// Mitsubishi GX Works2 project: BookEX6_14 Bistable   PLC: Q13UDV

// global labels: Global
VAR_GLOBAL
  bVar0 AT M5000 : BOOL;
  abArray0 AT M5010 : ARRAY [0..49] OF BOOL;
  sStr0 AT D5000 : STRING[199];
  sStr1 AT D5100 : STRING[199];
  sStr2 AT D5200 : STRING[199];
  sStr3 AT D5300 : STRING[199];
  sStr4 AT D5400 : STRING[199];
  sStr5 AT D5500 : STRING[199];
  sStr6 AT D5600 : STRING[199];
  sStr7 AT D5700 : STRING[199];
  sStr8 AT D5800 : STRING[199];
  sStr9 AT D5900 : STRING[199];
  iVar0 AT D4500 : INT;
  iVar1 AT D4501 : INT;
  iVar2 AT D4502 : INT;
  iVar3 AT D4503 : INT;
  iVar4 AT D4504 : INT;
  iVar5 AT D4505 : INT;
  iVar6 AT D4506 : INT;
  iVar7 AT D4507 : INT;
  iVar8 AT D4508 : INT;
  iVar9 AT D4509 : INT;
  dVar0 AT D4510 : DINT;
  dVar1 AT D4512 : DINT;
  dVar2 AT D4514 : DINT;
  dVar3 AT D4516 : DINT;
  dVar4 AT D4518 : DINT;
  dVar5 AT D4520 : DINT;
  dVar6 AT D4522 : DINT;
  dVar7 AT D4524 : DINT;
  dVar8 AT D4526 : DINT;
  dVar9 AT D4528 : DINT;
  wVar0 AT D4530 : WORD;
  wVar1 AT D4531 : WORD;
  wVar2 AT D4532 : WORD;
  wVar3 AT D4533 : WORD;
  wVar4 AT D4534 : WORD;
  wVar5 AT D4535 : WORD;
  wVar6 AT D4536 : WORD;
  wVar7 AT D4537 : WORD;
  wVar8 AT D4538 : WORD;
  wVar9 AT D4539 : WORD;
  dwVar0 AT D4540 : DWORD;
  dwVar1 AT D4542 : DWORD;
  dwVar2 AT D4544 : DWORD;
  dwVar3 AT D4546 : DWORD;
  dwVar4 AT D4548 : DWORD;
  dwVar5 AT D4550 : DWORD;
  dwVar6 AT D4552 : DWORD;
  dwVar7 AT D4554 : DWORD;
  dwVar8 AT D4556 : DWORD;
  dwVar9 AT D4558 : DWORD;
  fsVar0 AT D4560 : REAL;
  fsVar1 AT D4562 : REAL;
  fsVar2 AT D4564 : REAL;
  fsVar3 AT D4566 : REAL;
  fsVar4 AT D4568 : REAL;
  fsVar5 AT D4570 : REAL;
  fsVar6 AT D4572 : REAL;
  fsVar7 AT D4574 : REAL;
  fsVar8 AT D4576 : REAL;
  fsVar9 AT D4578 : REAL;
  fdVar0 AT D4580 : LREAL;
  tTime0 AT D4620 : TIME;
  tTime1 AT D4622 : TIME;
  tTime2 AT D4624 : TIME;
  tTime3 AT D4626 : TIME;
  tTime4 AT D4628 : TIME;
  tTime5 AT D4630 : TIME;
  tTime6 AT D4632 : TIME;
  tTime7 AT D4634 : TIME;
  tTime8 AT D4636 : TIME;
  tTime9 AT D4638 : TIME;
  tTime10 AT D4640 : TIME;
  bVar1 AT M5001 : BOOL;
  bVar2 AT M5002 : BOOL;
  bVar3 AT M5003 : BOOL;
  bVar4 AT M5004 : BOOL;
  bVar5 AT M5005 : BOOL;
  bVar6 AT M5006 : BOOL;
  bVar7 AT M5007 : BOOL;
  bVar8 AT M5008 : BOOL;
  bVar9 AT M5009 : BOOL;
  abArray1 AT M5060 : ARRAY [0..49] OF BOOL;
  abArray2 AT M5110 : ARRAY [0..49] OF BOOL;
  abArray3 AT M5160 : ARRAY [0..49] OF BOOL;
  abArray4 AT M5210 : ARRAY [0..49] OF BOOL;
  abArray5 AT M5260 : ARRAY [0..49] OF BOOL;
  abArray6 AT M5310 : ARRAY [0..49] OF BOOL;
  abArray7 AT M5360 : ARRAY [0..49] OF BOOL;
  abArray8 AT M5410 : ARRAY [0..49] OF BOOL;
  abArray9 AT M5460 : ARRAY [0..49] OF BOOL;
  fdVar1 AT D4584 : LREAL;
  fdVar2 AT D4588 : LREAL;
  fdVar3 AT D4592 : LREAL;
  fdVar4 AT D4596 : LREAL;
  fdVar5 AT D4600 : LREAL;
  fdVar6 AT D4604 : LREAL;
  fdVar7 AT D4608 : LREAL;
  fdVar8 AT D4612 : LREAL;
  fdVar9 AT D4616 : LREAL;
  aSendData1 AT D100 : ARRAY [0..9] OF INT;
  aiTxData AT D4000 : ARRAY [0..99] OF INT;
  aiRxData AT D4100 : ARRAY [0..99] OF INT;
  iOpenOK AT D3900 : INT;
  iOpenERR AT D3901 : INT;
  iSendOK AT D3902 : INT;
  iSendERR AT D3903 : INT;
  iCloseOK AT D3906 : INT;
  iCloseERR AT D3907 : INT;
  iRecvOK AT D3904 : INT;
  iRecvERR AT D3905 : INT;
  aiTxData2 AT D4200 : ARRAY [0..99] OF INT;
  aiRxData2 AT D4300 : ARRAY [0..99] OF INT;
  iOpenOK2 AT D3908 : INT;
  iOpenERR2 AT D3909 : INT;
  iSendOK2 AT D3910 : INT;
  iSendERR2 AT D3911 : INT;
  iRecvOK2 AT D3912 : INT;
  iRecvERR2 AT D3913 : INT;
  iCloseOK2 AT D3914 : INT;
  iCloseERR2 AT D3915 : INT;
  iEOpenComp AT D3916 : INT;
  iEOpenReq AT D3917 : INT;
  iERecvFlag AT D3918 : INT;
  iOpenCode AT D3919 : INT;
  iSendCode AT D3920 : INT;
  iRecvCode AT D3921 : INT;
  iCloseCode AT D3922 : INT;
  iOpenCode2 AT D3923 : INT;
  iSendCode2 AT D3924 : INT;
  iRecvCode2 AT D3925 : INT;
  iCloseCode2 AT D3926 : INT;
  aRecvData1 AT D110 : ARRAY [0..9] OF INT;
  aSendData2 AT D120 : ARRAY [0..9] OF INT;
  aRecvData2 AT D130 : ARRAY [0..9] OF INT;
END_VAR
// user libraries (not included): HMI

FUNCTION_BLOCK BiRS
VAR_INPUT
  b_S : BOOL;
  b_R : BOOL;
END_VAR
VAR_OUTPUT
  b_Q : BOOL;
END_VAR
;
b_Q := (b_Q OR b_S) AND NOT b_R;
END_FUNCTION_BLOCK

FUNCTION_BLOCK BiSR
VAR_INPUT
  b_S : BOOL;
  b_R : BOOL;
END_VAR
VAR_OUTPUT
  b_Q : BOOL;
END_VAR
;
b_Q := b_S OR (b_Q AND NOT b_R);
END_FUNCTION_BLOCK

FUNCTION_BLOCK D_FF
VAR_INPUT
  b_SET : BOOL;
  b_D : BOOL;
  b_CK : BOOL;
  b_RST : BOOL;
END_VAR
VAR_OUTPUT
  b_Q : BOOL;
END_VAR
VAR
  oldCK : BOOL;
END_VAR
;
IF b_RST OR b_SET THEN
	b_Q := NOT b_RST;
ELSIF b_CK AND NOT oldCK THEN
	b_Q := b_D;
END_IF;
oldCK := b_CK;
END_FUNCTION_BLOCK

FUNCTION_BLOCK EdgeTrigLD
VAR_INPUT
  b_C : BOOL;
END_VAR
VAR_OUTPUT
  b_F : BOOL;
  b_X : BOOL;
END_VAR
(* structured ladder/FBD written out as ST: instructions are called as NAME(EN, inputs, outputs); _pN, _eN, _tN stand for wires *)
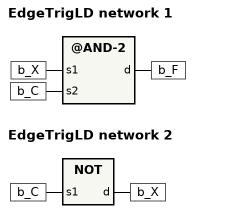
(* network 1 *)
b_F := @AND-2(b_X, b_C);
(* network 2 *)
b_X := NOT(b_C);
END_FUNCTION_BLOCK

FUNCTION_BLOCK EdgeTrigST
VAR_INPUT
  b_C : BOOL;
END_VAR
VAR_OUTPUT
  b_F : BOOL;
END_VAR
VAR
  oldC : BOOL;
END_VAR
;
IF b_C AND NOT oldC THEN
	b_F := TRUE;
ELSE
	b_F := FALSE;
END_IF;
oldC := b_C;
END_FUNCTION_BLOCK

FUNCTION_BLOCK JK_FF
VAR_INPUT
  b_SET : BOOL;
  b_J : BOOL;
  b_CK : BOOL;
END_VAR
VAR_OUTPUT
  b_Q : BOOL;
END_VAR
VAR_INPUT
  b_RST : BOOL;
END_VAR
VAR
  oldCK : BOOL;
END_VAR
VAR_INPUT
  b_K : BOOL;
END_VAR
;
IF b_RST OR b_SET THEN
	b_Q := NOT b_RST;
ELSIF b_CK AND NOT oldCK THEN
	IF b_J XOR b_K THEN 
		b_Q := b_J;
	ELSE 
		b_Q := b_K XOR b_Q;
	END_IF;
END_IF;
oldCK := b_CK;
END_FUNCTION_BLOCK

FUNCTION_BLOCK JoySw
VAR_INPUT
  SwX1 : BOOL;
END_VAR
VAR_OUTPUT
  LampY1 : BOOL;
END_VAR
VAR_INPUT
  SwX2 : BOOL;
END_VAR
VAR_OUTPUT
  LampY2 : BOOL;
  LampY3 : BOOL;
  LampY4 : BOOL;
END_VAR
VAR_INPUT
  SwX3 : BOOL;
  SwX4 : BOOL;
  Reset : BOOL;
END_VAR
VAR_OUTPUT
  LampY5 : BOOL;
END_VAR
VAR_INPUT
  SwX5 : BOOL;
  SwX6 : BOOL;
  SwX7 : BOOL;
  SwX8 : BOOL;
END_VAR
VAR_OUTPUT
  LampY6 : BOOL;
  LampY7 : BOOL;
  LampY8 : BOOL;
  LampR : BOOL;
END_VAR
(* structured ladder/FBD written out as ST: instructions are called as NAME(EN, inputs, outputs); _pN, _eN, _tN stand for wires *)
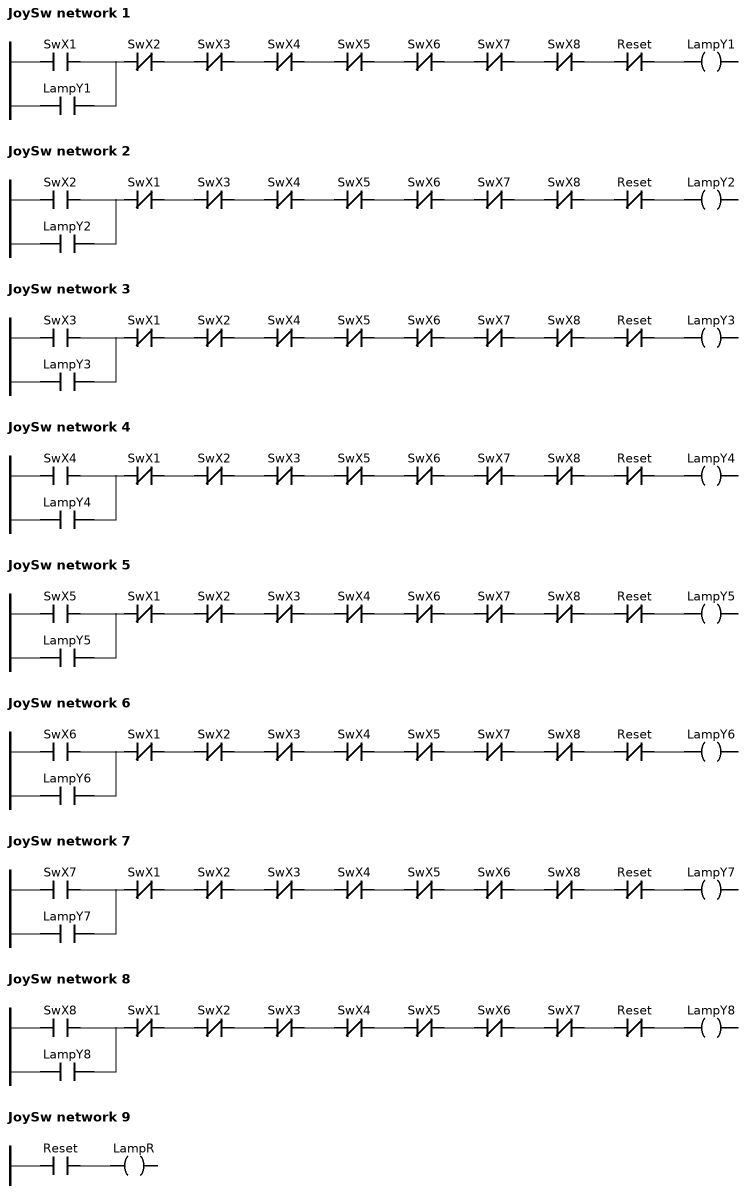
(* network 1 *)
LampY1 := ((((((((SwX1 OR LampY1) AND NOT SwX2) AND NOT SwX3) AND NOT SwX4) AND NOT SwX5) AND NOT SwX6) AND NOT SwX7) AND NOT SwX8) AND NOT Reset;
(* network 2 *)
LampY2 := ((((((((SwX2 OR LampY2) AND NOT SwX1) AND NOT SwX3) AND NOT SwX4) AND NOT SwX5) AND NOT SwX6) AND NOT SwX7) AND NOT SwX8) AND NOT Reset;
(* network 3 *)
LampY3 := ((((((((SwX3 OR LampY3) AND NOT SwX1) AND NOT SwX2) AND NOT SwX4) AND NOT SwX5) AND NOT SwX6) AND NOT SwX7) AND NOT SwX8) AND NOT Reset;
(* network 4 *)
LampY4 := ((((((((SwX4 OR LampY4) AND NOT SwX1) AND NOT SwX2) AND NOT SwX3) AND NOT SwX5) AND NOT SwX6) AND NOT SwX7) AND NOT SwX8) AND NOT Reset;
(* network 5 *)
LampY5 := ((((((((SwX5 OR LampY5) AND NOT SwX1) AND NOT SwX2) AND NOT SwX3) AND NOT SwX4) AND NOT SwX6) AND NOT SwX7) AND NOT SwX8) AND NOT Reset;
(* network 6 *)
LampY6 := ((((((((SwX6 OR LampY6) AND NOT SwX1) AND NOT SwX2) AND NOT SwX3) AND NOT SwX4) AND NOT SwX5) AND NOT SwX7) AND NOT SwX8) AND NOT Reset;
(* network 7 *)
LampY7 := ((((((((SwX7 OR LampY7) AND NOT SwX1) AND NOT SwX2) AND NOT SwX3) AND NOT SwX4) AND NOT SwX5) AND NOT SwX6) AND NOT SwX8) AND NOT Reset;
(* network 8 *)
LampY8 := ((((((((SwX8 OR LampY8) AND NOT SwX1) AND NOT SwX2) AND NOT SwX3) AND NOT SwX4) AND NOT SwX5) AND NOT SwX6) AND NOT SwX7) AND NOT Reset;
(* network 9 *)
LampR := Reset;
END_FUNCTION_BLOCK

FUNCTION_BLOCK Latch
VAR_INPUT
  b_D : BOOL;
  b_L : BOOL;
  b_R : BOOL;
END_VAR
VAR_OUTPUT
  b_Q : BOOL;
END_VAR
;
IF b_R THEN				 
	b_Q := FALSE;
ELSIF b_L THEN		 
	b_Q := b_D;
END_IF;
END_FUNCTION_BLOCK

FUNCTION_BLOCK LockSw
VAR_INPUT
  SwX1 : BOOL;
END_VAR
VAR_OUTPUT
  LampY1 : BOOL;
END_VAR
VAR_INPUT
  SwX2 : BOOL;
END_VAR
VAR_OUTPUT
  LampY2 : BOOL;
END_VAR
(* structured ladder/FBD written out as ST: instructions are called as NAME(EN, inputs, outputs); _pN, _eN, _tN stand for wires *)
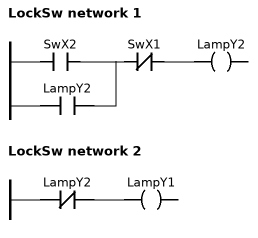
(* network 1 *)
LampY2 := (SwX2 OR LampY2) AND NOT SwX1;
(* network 2 *)
LampY1 := NOT LampY2;
END_FUNCTION_BLOCK

FUNCTION_BLOCK ModeSw
VAR_INPUT
  SwL : BOOL;
  SwR : BOOL;
END_VAR
VAR_OUTPUT
  LampY1 : BOOL;
  LampY2 : BOOL;
END_VAR
VAR
  iMode : INT;
END_VAR
VAR_OUTPUT
  i_Mode : INT;
END_VAR
;
IF LDP(TRUE, SwL)  THEN
	IF iMode = 0 THEN
		iMode := 1;
	ELSIF iMode = 2 THEN
		iMode := 0;
	END_IF;
END_IF;
IF LDP(TRUE, SwR)  THEN
	IF iMode = 1 THEN
		iMode := 0;
	ELSIF iMode = 0 THEN
		iMode := 2;
	END_IF;
END_IF;
LampY1 := INT_TO_WORD(iMode) = 1;
LampY2 := INT_TO_WORD(iMode) = 2;
i_Mode := iMode;
END_FUNCTION_BLOCK

FUNCTION_BLOCK NAND_ESR
VAR_INPUT
  b_S : BOOL;
END_VAR
VAR_OUTPUT
  b_Q : BOOL;
  b_nQ : BOOL;
END_VAR
VAR
  bS : BOOL;
  bR : BOOL;
END_VAR
VAR_INPUT
  b_R : BOOL;
  b_En : BOOL;
END_VAR
(* structured ladder/FBD written out as ST: instructions are called as NAME(EN, inputs, outputs); _pN, _eN, _tN stand for wires *)
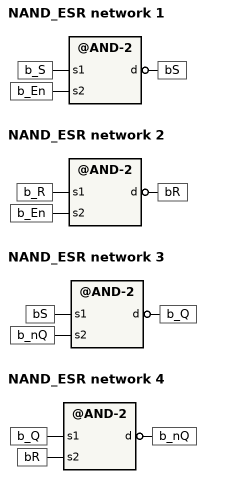
(* network 1 *)
bS := NOT (@AND-2(b_S, b_En));
(* network 2 *)
bR := NOT (@AND-2(b_R, b_En));
(* network 3 *)
b_Q := NOT (@AND-2(bS, b_nQ));
(* network 4 *)
b_nQ := NOT (@AND-2(b_Q, bR));
END_FUNCTION_BLOCK

FUNCTION_BLOCK NAND_SR
VAR_INPUT
  b_R : BOOL;
END_VAR
VAR_OUTPUT
  b_Q : BOOL;
  b_nQ : BOOL;
END_VAR
VAR_INPUT
  b_S : BOOL;
END_VAR
(* structured ladder/FBD written out as ST: instructions are called as NAME(EN, inputs, outputs); _pN, _eN, _tN stand for wires *)
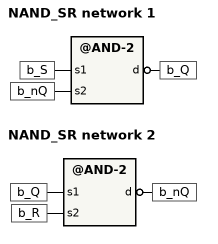
(* network 1 *)
b_Q := NOT (@AND-2(b_S, b_nQ));
(* network 2 *)
b_nQ := NOT (@AND-2(b_Q, b_R));
END_FUNCTION_BLOCK

FUNCTION_BLOCK NOR_ESR
VAR_INPUT
  b_R : BOOL;
  b_S : BOOL;
END_VAR
VAR_OUTPUT
  b_Q : BOOL;
  b_nQ : BOOL;
END_VAR
VAR_INPUT
  b_En : BOOL;
END_VAR
VAR
  bR : BOOL;
  bS : BOOL;
END_VAR
(* structured ladder/FBD written out as ST: instructions are called as NAME(EN, inputs, outputs); _pN, _eN, _tN stand for wires *)
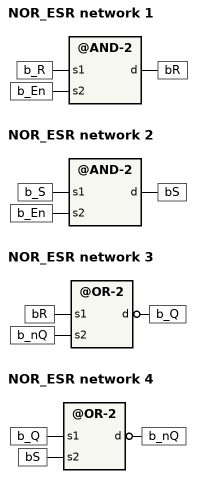
(* network 1 *)
bR := @AND-2(b_R, b_En);
(* network 2 *)
bS := @AND-2(b_S, b_En);
(* network 3 *)
b_Q := NOT (@OR-2(bR, b_nQ));
(* network 4 *)
b_nQ := NOT (@OR-2(b_Q, bS));
END_FUNCTION_BLOCK

FUNCTION_BLOCK NOR_SR
VAR_INPUT
  b_R : BOOL;
  b_S : BOOL;
END_VAR
VAR_OUTPUT
  b_Q : BOOL;
  b_nQ : BOOL;
END_VAR
(* structured ladder/FBD written out as ST: instructions are called as NAME(EN, inputs, outputs); _pN, _eN, _tN stand for wires *)
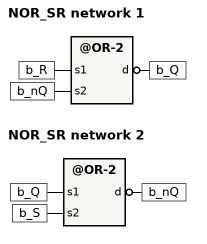
(* network 1 *)
b_Q := NOT (@OR-2(b_R, b_nQ));
(* network 2 *)
b_nQ := NOT (@OR-2(b_Q, b_S));
END_FUNCTION_BLOCK

FUNCTION_BLOCK PianoSw
VAR_INPUT
  SwX1 : BOOL;
END_VAR
VAR_OUTPUT
  LampY1 : BOOL;
END_VAR
VAR_INPUT
  SwX2 : BOOL;
END_VAR
VAR_OUTPUT
  LampY2 : BOOL;
  LampY3 : BOOL;
  LampY4 : BOOL;
END_VAR
VAR_INPUT
  SwX3 : BOOL;
  SwX4 : BOOL;
  Reset : BOOL;
END_VAR
VAR_OUTPUT
  LampY5 : BOOL;
END_VAR
(* structured ladder/FBD written out as ST: instructions are called as NAME(EN, inputs, outputs); _pN, _eN, _tN stand for wires *)
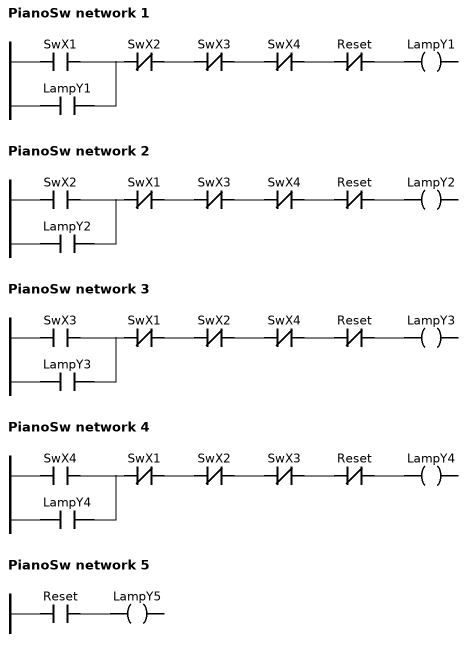
(* network 1 *)
LampY1 := ((((SwX1 OR LampY1) AND NOT SwX2) AND NOT SwX3) AND NOT SwX4) AND NOT Reset;
(* network 2 *)
LampY2 := ((((SwX2 OR LampY2) AND NOT SwX1) AND NOT SwX3) AND NOT SwX4) AND NOT Reset;
(* network 3 *)
LampY3 := ((((SwX3 OR LampY3) AND NOT SwX1) AND NOT SwX2) AND NOT SwX4) AND NOT Reset;
(* network 4 *)
LampY4 := ((((SwX4 OR LampY4) AND NOT SwX1) AND NOT SwX2) AND NOT SwX3) AND NOT Reset;
(* network 5 *)
LampY5 := Reset;
END_FUNCTION_BLOCK

FUNCTION_BLOCK RS_FF
VAR_INPUT
  b_S : BOOL;
  b_R : BOOL;
  b_RST : BOOL;
END_VAR
VAR_OUTPUT
  b_Q : BOOL;
END_VAR
VAR_INPUT
  b_SET : BOOL;
  b_CK : BOOL;
END_VAR
VAR
  oldCK : BOOL;
END_VAR
;
IF b_RST OR b_SET THEN
	b_Q := NOT b_RST;
ELSIF b_CK AND NOT oldCK THEN
	IF b_R THEN
		b_Q := FALSE;
	ELSIF b_S THEN
		b_Q := TRUE;
	END_IF;
END_IF;
oldCK := b_CK;
END_FUNCTION_BLOCK

FUNCTION_BLOCK RS_FF2
VAR_INPUT
  b_S : BOOL;
  b_R : BOOL;
  b_RST : BOOL;
END_VAR
VAR_OUTPUT
  b_Q : BOOL;
END_VAR
VAR
  oldS : BOOL;
  oldR : BOOL;
END_VAR
VAR_INPUT
  b_SET : BOOL;
END_VAR
;
IF b_RST OR b_SET THEN
	b_Q := NOT b_RST;
ELSIF b_R AND NOT oldR THEN
	b_Q := FALSE;
ELSIF b_S AND NOT oldS THEN
	b_Q := TRUE;
END_IF;

oldS := b_S;
oldR := b_R;
END_FUNCTION_BLOCK

FUNCTION_BLOCK SelSw
VAR_INPUT
  SwX1 : BOOL;
END_VAR
VAR_OUTPUT
  LampY1 : BOOL;
END_VAR
VAR_INPUT
  SwX2 : BOOL;
END_VAR
VAR_OUTPUT
  LampY2 : BOOL;
END_VAR
VAR_IN_OUT
  SelData : INT;
END_VAR
(* structured ladder/FBD written out as ST: instructions are called as NAME(EN, inputs, outputs); _pN, _eN, _tN stand for wires *)
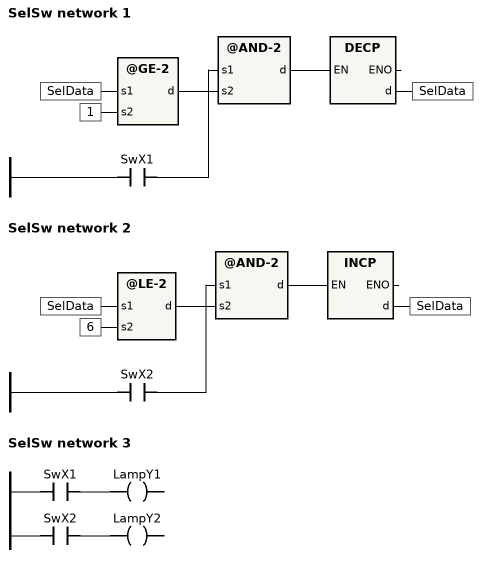
(* network 1 *)
DECP(@AND-2(SwX1, @GE-2(SelData, 1)), SelData);
(* network 2 *)
INCP(@AND-2(SwX2, @LE-2(SelData, 6)), SelData);
(* network 3 *)
LampY1 := SwX1;
LampY2 := SwX2;
END_FUNCTION_BLOCK

FUNCTION_BLOCK T_FF
VAR_INPUT
  b_T : BOOL;
  b_CK : BOOL;
  b_RST : BOOL;
END_VAR
VAR_OUTPUT
  b_Q : BOOL;
END_VAR
VAR
  oldCK : BOOL;
END_VAR
;
IF b_RST THEN
	b_Q := FALSE;
ELSIF b_CK AND NOT oldCK THEN
	IF b_T THEN b_Q := NOT b_Q; END_IF;
END_IF;
oldCK := b_CK;
END_FUNCTION_BLOCK

FUNCTION_BLOCK ToggSw
VAR_INPUT
  SwX : BOOL;
END_VAR
VAR_OUTPUT
  LampY : BOOL;
END_VAR
(* structured ladder/FBD written out as ST: instructions are called as NAME(EN, inputs, outputs); _pN, _eN, _tN stand for wires *)
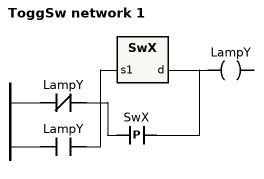
(* network 1 *)
(* element kind 19 SwX <- LampY *)
LampY := (NOT LampY AND LDP(TRUE, SwX)) OR _feedback;
END_FUNCTION_BLOCK

PROGRAM ExD_FF
VAR
  D_FF_1 : D_FF;
  HMI05_1 : HMI05;
END_VAR
(* structured ladder/FBD written out as ST: instructions are called as NAME(EN, inputs, outputs); _pN, _eN, _tN stand for wires *)
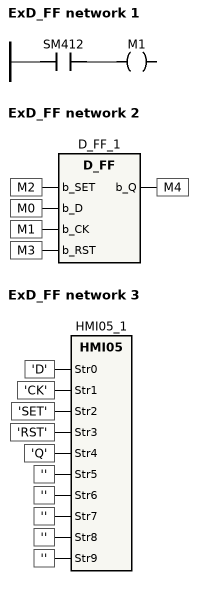
(* network 1 *)
M1 := SM412;
(* network 2 *)
D_FF_1(b_SET := M2, b_D := M0, b_CK := M1, b_RST := M3, b_Q => M4);
(* network 3 *)
HMI05_1(Str0 := 'D', Str1 := 'CK', Str2 := 'SET', Str3 := 'RST', Str4 := 'Q', Str5 := '', Str6 := '', Str7 := '', Str8 := '', Str9 := '');
END_PROGRAM

PROGRAM ExJK_FF
VAR
  JK_FF_1 : JK_FF;
  HMI05_1 : HMI05;
END_VAR
(* structured ladder/FBD written out as ST: instructions are called as NAME(EN, inputs, outputs); _pN, _eN, _tN stand for wires *)
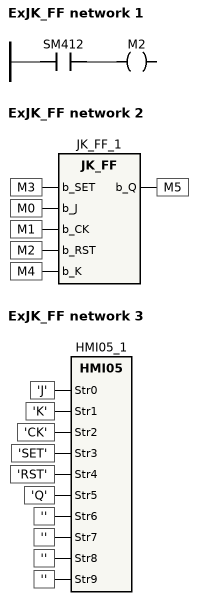
(* network 1 *)
M2 := SM412;
(* network 2 *)
JK_FF_1(b_SET := M3, b_J := M0, b_CK := M1, b_RST := M2, b_K := M4, b_Q => M5);
(* network 3 *)
HMI05_1(Str0 := 'J', Str1 := 'K', Str2 := 'CK', Str3 := 'SET', Str4 := 'RST', Str5 := 'Q', Str6 := '', Str7 := '', Str8 := '', Str9 := '');
END_PROGRAM

PROGRAM ExLatch
VAR
  NOR_SR_1 : NOR_SR;
  NAND_SR_1 : NAND_SR;
  HMI05_1 : HMI05;
END_VAR
(* structured ladder/FBD written out as ST: instructions are called as NAME(EN, inputs, outputs); _pN, _eN, _tN stand for wires *)
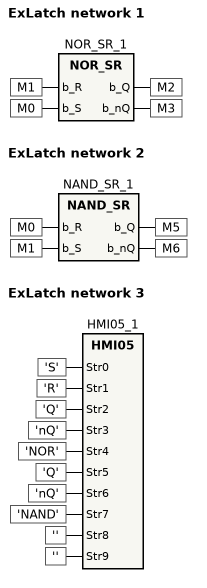
(* network 1 *)
NOR_SR_1(b_R := M1, b_S := M0, b_Q => M2, b_nQ => M3);
(* network 2 *)
NAND_SR_1(b_R := M0, b_S := M1, b_Q => M5, b_nQ => M6);
(* network 3 *)
HMI05_1(Str0 := 'S', Str1 := 'R', Str2 := 'Q', Str3 := 'nQ', Str4 := 'NOR', Str5 := 'Q', Str6 := 'nQ', Str7 := 'NAND', Str8 := '', Str9 := '');
END_PROGRAM

PROGRAM ExLatch2
VAR
  NOR_ESR_1 : NOR_ESR;
  NAND_ESR_1 : NAND_ESR;
  HMI05_1 : HMI05;
END_VAR
(* structured ladder/FBD written out as ST: instructions are called as NAME(EN, inputs, outputs); _pN, _eN, _tN stand for wires *)
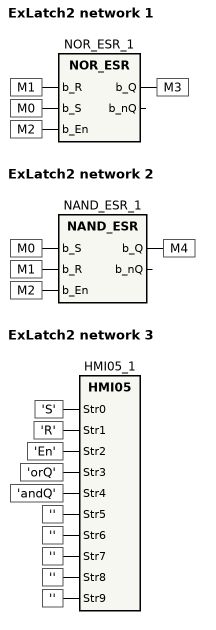
(* network 1 *)
NOR_ESR_1(b_R := M1, b_S := M0, b_En := M2, b_Q => M3);
(* network 2 *)
NAND_ESR_1(b_S := M0, b_R := M1, b_En := M2, b_Q => M4);
(* network 3 *)
HMI05_1(Str0 := 'S', Str1 := 'R', Str2 := 'En', Str3 := 'orQ', Str4 := 'andQ', Str5 := '', Str6 := '', Str7 := '', Str8 := '', Str9 := '');
END_PROGRAM

PROGRAM ExRS
VAR
  RS_E_1 : RS_E;
  BiRS_1 : BiRS;
  HMI05_1 : HMI05;
END_VAR
(* structured ladder/FBD written out as ST: instructions are called as NAME(EN, inputs, outputs); _pN, _eN, _tN stand for wires *)
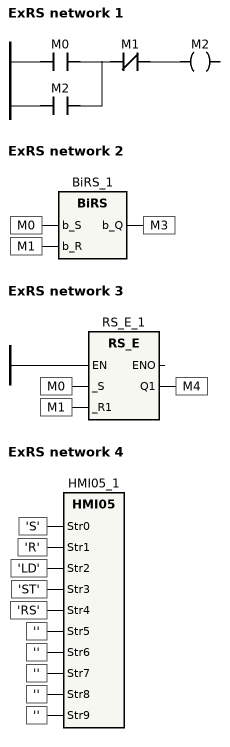
(* network 1 *)
M2 := (M0 OR M2) AND NOT M1;
(* network 2 *)
BiRS_1(b_S := M0, b_R := M1, b_Q => M3);
(* network 3 *)
RS_E_1(EN := TRUE, _S := M0, _R1 := M1, Q1 => M4);
(* network 4 *)
HMI05_1(Str0 := 'S', Str1 := 'R', Str2 := 'LD', Str3 := 'ST', Str4 := 'RS', Str5 := '', Str6 := '', Str7 := '', Str8 := '', Str9 := '');
END_PROGRAM

PROGRAM ExRS_FF
VAR
  RS_FF_1 : RS_FF;
  HMI05_1 : HMI05;
END_VAR
(* structured ladder/FBD written out as ST: instructions are called as NAME(EN, inputs, outputs); _pN, _eN, _tN stand for wires *)
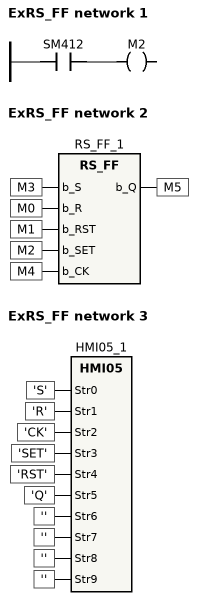
(* network 1 *)
M2 := SM412;
(* network 2 *)
RS_FF_1(b_S := M3, b_R := M0, b_RST := M1, b_SET := M2, b_CK := M4, b_Q => M5);
(* network 3 *)
HMI05_1(Str0 := 'S', Str1 := 'R', Str2 := 'CK', Str3 := 'SET', Str4 := 'RST', Str5 := 'Q', Str6 := '', Str7 := '', Str8 := '', Str9 := '');
END_PROGRAM

PROGRAM ExSR
VAR
  SR_E_1 : SR_E;
  RS_E_1 : RS_E;
  BiSR_1 : BiSR;
  HMI05_1 : HMI05;
END_VAR
(* structured ladder/FBD written out as ST: instructions are called as NAME(EN, inputs, outputs); _pN, _eN, _tN stand for wires *)
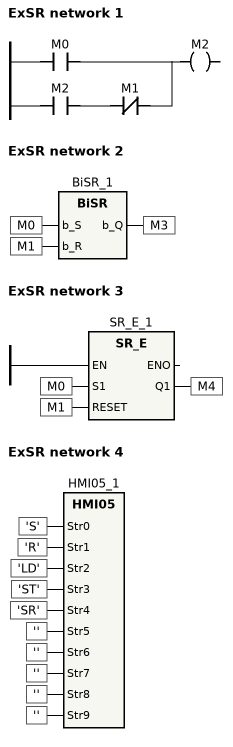
(* network 1 *)
M2 := M0 OR (M2 AND NOT M1);
(* network 2 *)
BiSR_1(b_S := M0, b_R := M1, b_Q => M3);
(* network 3 *)
SR_E_1(EN := TRUE, S1 := M0, RESET := M1, Q1 => M4);
(* network 4 *)
HMI05_1(Str0 := 'S', Str1 := 'R', Str2 := 'LD', Str3 := 'ST', Str4 := 'SR', Str5 := '', Str6 := '', Str7 := '', Str8 := '', Str9 := '');
END_PROGRAM

PROGRAM ExSwitch
VAR
  ToggSw_1 : ToggSw;
  LockSw_1 : LockSw;
  PianoSw_1 : PianoSw;
  SelSw_1 : SelSw;
  JoySw_1 : JoySw;
  ModeSw_1 : ModeSw;
END_VAR
(* structured ladder/FBD written out as ST: instructions are called as NAME(EN, inputs, outputs); _pN, _eN, _tN stand for wires *)
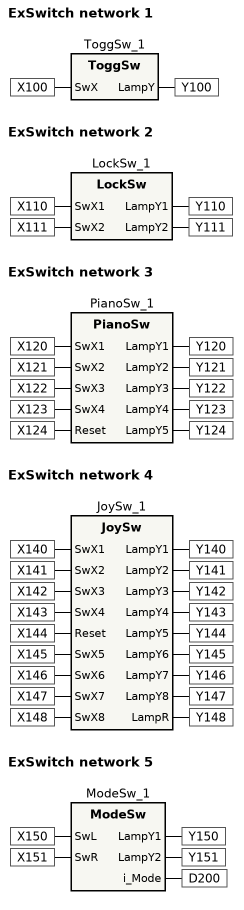
(* network 1 *)
ToggSw_1(SwX := X100, LampY => Y100);
(* network 2 *)
LockSw_1(SwX1 := X110, SwX2 := X111, LampY1 => Y110, LampY2 => Y111);
(* network 3 *)
PianoSw_1(SwX1 := X120, SwX2 := X121, SwX3 := X122, SwX4 := X123, Reset := X124, LampY1 => Y120, LampY2 => Y121, LampY3 => Y122, LampY4 => Y123, LampY5 => Y124);
(* network 4 *)
JoySw_1(SwX1 := X140, SwX2 := X141, SwX3 := X142, SwX4 := X143, Reset := X144, SwX5 := X145, SwX6 := X146, SwX7 := X147, SwX8 := X148, LampY1 => Y140, LampY2 => Y141, LampY3 => Y142, LampY4 => Y143, LampY5 => Y144, LampY6 => Y145, LampY7 => Y146, LampY8 => Y147, LampR => Y148);
(* network 5 *)
ModeSw_1(SwL := X150, SwR := X151, LampY1 => Y150, LampY2 => Y151, i_Mode => D200);
END_PROGRAM

PROGRAM ExT_FF
VAR
  T_FF_1 : T_FF;
  HMI05_1 : HMI05;
END_VAR
(* structured ladder/FBD written out as ST: instructions are called as NAME(EN, inputs, outputs); _pN, _eN, _tN stand for wires *)
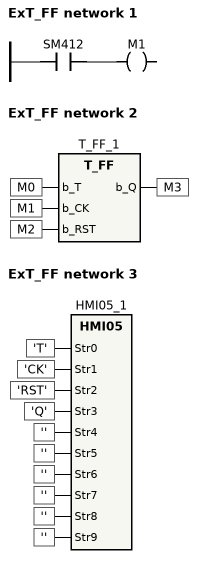
(* network 1 *)
M1 := SM412;
(* network 2 *)
T_FF_1(b_T := M0, b_CK := M1, b_RST := M2, b_Q => M3);
(* network 3 *)
HMI05_1(Str0 := 'T', Str1 := 'CK', Str2 := 'RST', Str3 := 'Q', Str4 := '', Str5 := '', Str6 := '', Str7 := '', Str8 := '', Str9 := '');
END_PROGRAM

PROGRAM ExRS2
VAR
  RS_E_1 : RS_E;
  HMI05_1 : HMI05;
  RS_E_2 : RS_E;
  RS_E_3 : RS_E;
  HMI05_2 : HMI05;
END_VAR
(* structured ladder/FBD written out as ST: instructions are called as NAME(EN, inputs, outputs); _pN, _eN, _tN stand for wires *)
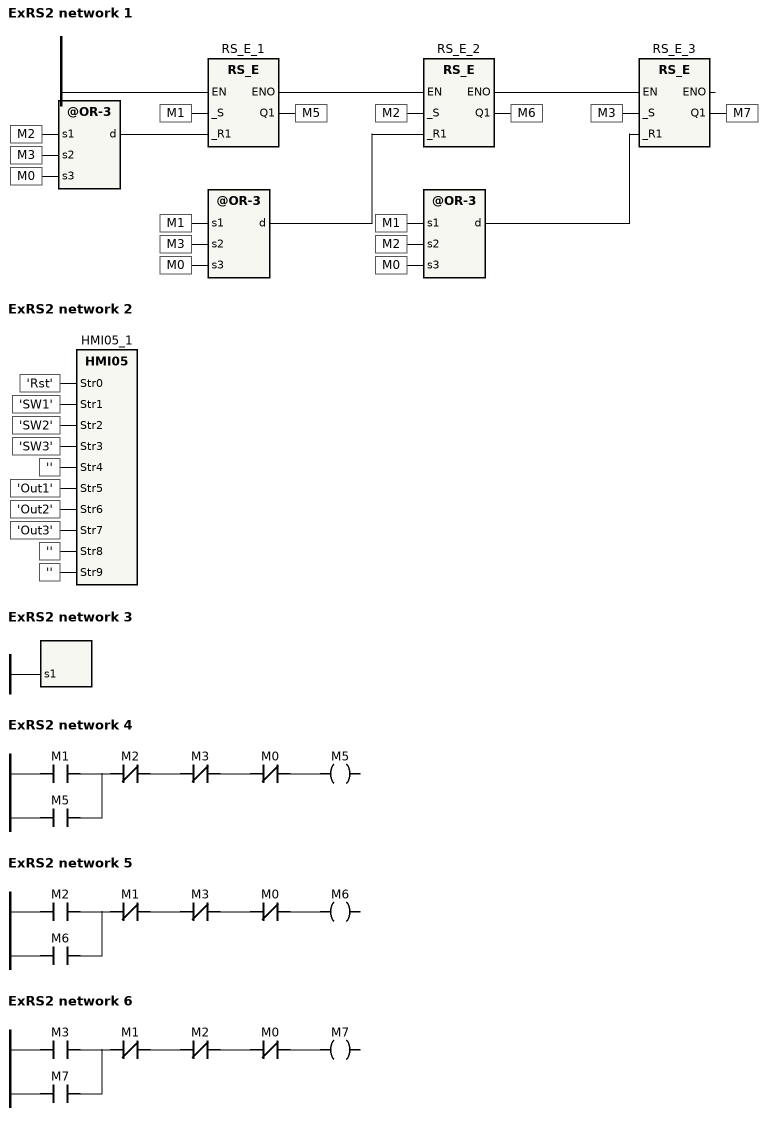
(* network 1 *)
RS_E_1(EN := TRUE, _S := M1, _R1 := @OR-3(M2, M3, M0), Q1 => M5);
RS_E_2(EN := RS_E_1.ENO, _S := M2, _R1 := @OR-3(M1, M3, M0), Q1 => M6);
RS_E_3(EN := RS_E_2.ENO, _S := M3, _R1 := @OR-3(M1, M2, M0), Q1 => M7);
(* network 2 *)
HMI05_1(Str0 := 'Rst', Str1 := 'SW1', Str2 := 'SW2', Str3 := 'SW3', Str4 := '', Str5 := 'Out1', Str6 := 'Out2', Str7 := 'Out3', Str8 := '', Str9 := '');
(* network 3 *)
(* element kind 10  <- TRUE *)
(* network 4 *)
M5 := (((M1 OR M5) AND NOT M2) AND NOT M3) AND NOT M0;
(* network 5 *)
M6 := (((M2 OR M6) AND NOT M1) AND NOT M3) AND NOT M0;
(* network 6 *)
M7 := (((M3 OR M7) AND NOT M1) AND NOT M2) AND NOT M0;
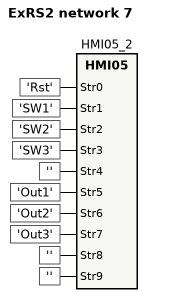
(* network 7 *)
HMI05_2(Str0 := 'Rst', Str1 := 'SW1', Str2 := 'SW2', Str3 := 'SW3', Str4 := '', Str5 := 'Out1', Str6 := 'Out2', Str7 := 'Out3', Str8 := '', Str9 := '');
END_PROGRAM

PROGRAM ExRS3
VAR
  RS_E_1 : RS_E;
  HMI05_1 : HMI05;
  HMI05_2 : HMI05;
END_VAR
(* structured ladder/FBD written out as ST: instructions are called as NAME(EN, inputs, outputs); _pN, _eN, _tN stand for wires *)
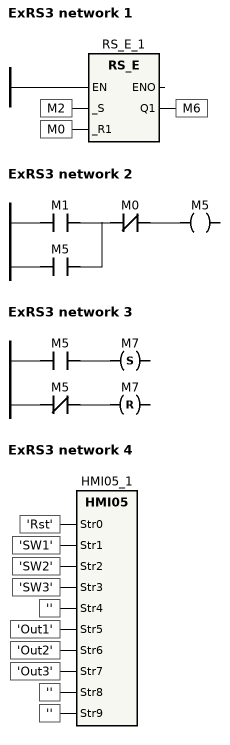
(* network 1 *)
RS_E_1(EN := TRUE, _S := M2, _R1 := M0, Q1 => M6);
(* network 2 *)
M5 := (M1 OR M5) AND NOT M0;
(* network 3 *)
SET(M5, M7);
RST(NOT M5, M7);
(* network 4 *)
HMI05_1(Str0 := 'Rst', Str1 := 'SW1', Str2 := 'SW2', Str3 := 'SW3', Str4 := '', Str5 := 'Out1', Str6 := 'Out2', Str7 := 'Out3', Str8 := '', Str9 := '');
END_PROGRAM

FUNCTION Bit2Word
VAR_INPUT
  Bit0 : BOOL;
  Bit1 : BOOL;
  Bit2 : BOOL;
  Bit3 : BOOL;
  Bit4 : BOOL;
  Bit5 : BOOL;
  Bit6 : BOOL;
  Bit7 : BOOL;
END_VAR
			
Bit2Word := SHL(SHL(SHL(SHL(SHL(SHL(SHL(BOOL_TO_WORD(Bit7),1) OR BOOL_TO_WORD(Bit6),1) 
                     OR BOOL_TO_WORD(Bit5),1) OR BOOL_TO_WORD(Bit4),1)
	                 OR BOOL_TO_WORD(Bit3),1) OR BOOL_TO_WORD(Bit2),1) 
	                 OR BOOL_TO_WORD(Bit1),1) OR BOOL_TO_WORD(Bit0);
END_FUNCTION

FUNCTION_BLOCK Word2Bit
VAR_INPUT
  IN : WORD;
END_VAR
VAR_OUTPUT
  Bit0 : BOOL;
  Bit1 : BOOL;
  Bit2 : BOOL;
  Bit3 : BOOL;
  Bit4 : BOOL;
  Bit5 : BOOL;
  Bit6 : BOOL;
  Bit7 : BOOL;
END_VAR
 
Bit0 := WORD_TO_BOOL(IN AND 16#0001);
Bit1 := WORD_TO_BOOL(SHR(IN AND 16#0002 , 1));
Bit2 := WORD_TO_BOOL(SHR(IN AND 16#0004 , 2));
Bit3 := WORD_TO_BOOL(SHR(IN AND 16#0008 , 3));
Bit4 := WORD_TO_BOOL(SHR(IN AND 16#0010 , 4));
Bit5 := WORD_TO_BOOL(SHR(IN AND 16#0020 , 5));
Bit6 := WORD_TO_BOOL(SHR(IN AND 16#0040 , 6));
Bit7 := WORD_TO_BOOL(SHR(IN AND 16#0080 , 7));
END_FUNCTION_BLOCK

FUNCTION_BLOCK JoySw_ST
VAR_INPUT
  wSwX : WORD;
  Reset : BOOL;
END_VAR
VAR_OUTPUT
  wLampY : WORD;
  LampR : BOOL;
END_VAR
VAR
  wTmpX : WORD;
  ix : INT;
  wTmpY : WORD;
END_VAR
;
LampR := Reset;
IF LampR OR (wSwX = 0) THEN
	wLampY := 0;  
	RETURN;
END_IF;
wTmpX := wSwX;
wTmpY := 1;
FOR ix := 0 TO 7 DO 
	IF (wTmpX AND wTmpY) <> 0 THEN
		EXIT;
	END_IF;
	wTmpY := SHL(wTmpY,1);
END_FOR;
wLampY := wTmpY;
END_FUNCTION_BLOCK

PROGRAM ExJoySw_ST
VAR
  Word2Bit_1 : Word2Bit;
  JoySw_ST_1 : JoySw_ST;
END_VAR
(* structured ladder/FBD written out as ST: instructions are called as NAME(EN, inputs, outputs); _pN, _eN, _tN stand for wires *)
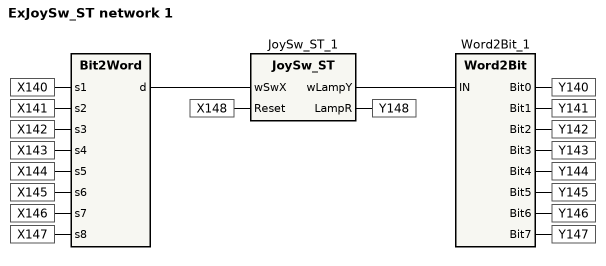
(* network 1 *)
JoySw_ST_1(wSwX := Bit2Word(X140, X141, X142, X143, X144, X145, X146, X147), Reset := X148, LampR => Y148);
Word2Bit_1(IN := JoySw_ST_1.wLampY, Bit0 => Y140, Bit1 => Y141, Bit2 => Y142, Bit3 => Y143, Bit4 => Y144, Bit5 => Y145, Bit6 => Y146, Bit7 => Y147);
END_PROGRAM

PROGRAM ExSR_ST
VAR
  fbErrLatch : SR;
  bErrorSensor : BOOL;
  bReset : BOOL;
  bSysError : BOOL;
  bLamp : BOOL;
  bResetSW : BOOL;
  SR_1 : SR;
END_VAR
;

(* 표준 SR 함수 블록 호출 및 파라미터 설정*)
fbErrLatch(
    _S1 := bErrorSensor,  	(* 에러를 감지하는  센서 입력 *)
    RESET  := bReset,    				(* 리셋 버튼을 누르면 에러 리셋 *)
    Q1 := bSysError   			(* 현재 에러 상태 Flag *)
);
 
IF bSysError THEN
    (*  Error가 발생하면 설비 중단 *)
    bLamp := TRUE;
END_IF;

IF bResetSW THEN
    (*  Reset 버튼이 ON되었을 때 처리 *)
    bErrorSensor := FALSE;
    bReset := TRUE;
ELSE
	bReset := FALSE;
END_IF;
END_PROGRAM

PROGRAM ExDFF
VAR
  HMI05_1 : HMI05;
END_VAR
(* structured ladder/FBD written out as ST: instructions are called as NAME(EN, inputs, outputs); _pN, _eN, _tN stand for wires *)
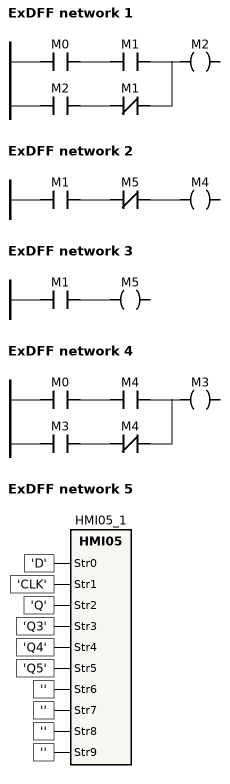
(* network 1 *)
M2 := (M0 AND M1) OR (M2 AND NOT M1);
(* network 2 *)
M4 := M1 AND NOT M5;
(* network 3 *)
M5 := M1;
(* network 4 *)
M3 := (M0 AND M4) OR (M3 AND NOT M4);
(* network 5 *)
HMI05_1(Str0 := 'D', Str1 := 'CLK', Str2 := 'Q', Str3 := 'Q3', Str4 := 'Q4', Str5 := 'Q5', Str6 := '', Str7 := '', Str8 := '', Str9 := '');
END_PROGRAM

PROGRAM ExJKFF
VAR
  HMI05_1 : HMI05;
END_VAR
(* structured ladder/FBD written out as ST: instructions are called as NAME(EN, inputs, outputs); _pN, _eN, _tN stand for wires *)
